FUNCTION ToRobotPoseSimple
VAR_INPUT
	x, y, theta : LREAL;
END_VAR
VAR
END_VAR
VAR_OUTPUT
	RobotPose : RobotPoseSimple;
END_VAR

RobotPose.x := x;
RobotPose.y := y;
RobotPose.theta := theta;

END_FUNCTION

(* stored: Version 1.1.0.1, ProductVersion 3.1.4024.11
   POU ToRobotPoseSimple: Id {d05a4df5-43b5-4944-96ea-d18cffe31b55}, SpecialFunc None *)
